# EPICS substitutions: si_ps_conv_fastcorrsApp/Db/crates.substitutions
file "sector.db"
{
    pattern { SEC }
            { 01 }
            { 02 }
            { 03 }
            { 04 }
            { 05 }
            { 06 }
            { 07 }
            { 08 }
            { 09 }
            { 10 }
            { 11 }
            { 12 }
            { 13 }
            { 14 }
            { 15 }
            { 16 }
            { 17 }
            { 19 }
            { 20 }
}
